// Mitsubishi GX Works2 project: ciclico   PLC: Q03UDV

PROGRAM MAIN
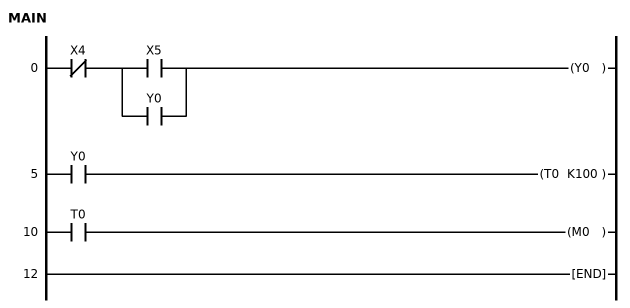
0     LDI     X4
      LD      X5
      OR      Y0
      ANB
      OUT     Y0
5     LD      Y0
      OUT     T0 K100
10    LD      T0
      OUT     M0
12    END
END_PROGRAM
